TYPE ST_AX5kIn :
STRUCT
	TorqueFeedbackIDN_S_84 		: INT;	(*Link To Process Data --> At--> IDN S-0-0084*)
	PositionFeedback1Value			: DINT;

END_STRUCT
END_TYPE

(* stored: Version 1.1.0.1, ProductVersion 3.1.4024.11
   DUT ST_AX5kIn: Id {75e1165f-23e5-4770-81b4-4035b883f56c} *)
